FUNCTION_BLOCK TestRecieve EXTENDS Object IMPLEMENTS IDataReciever
VAR
    buffer : testData;
    currentLength : UDINT;
END_VAR

{attribute '''NORMAL__COMMENT' := ' New data recieved'}
(* New data recieved*)
METHOD NewDataRecieved : HResult
VAR_INPUT
	data	: Data; //Data recieved
END_VAR
IF currentLength + data.length > 9999 THEN
    currentLength := 0;
END_IF

Tc2_System.MEMCPY(destAddr := ADR(buffer.buffer[currentLength]),srcAddr := data.data, n := data.length); 

currentLength := currentLength + data.length;
END_METHOD

(*Reset error, allways call super*)
METHOD Reset
Tc2_System.MEMSET(destAddr := ADR(buffer), fillByte := 0, n := SIZEOF(buffer));
currentLength := 0;
END_METHOD

END_FUNCTION_BLOCK

(* stored: Version 1.1.0.1, ProductVersion 3.1.4020.12
   POU TestRecieve: Id {ac45b7df-f119-44bf-ad93-44d7bc6f8a02}, SpecialFunc None
   Method NewDataRecieved: Id {5380409a-4052-40e4-9eb6-8bd6a2573e60}
   Method Reset: Id {546fd031-9c6c-4eaf-92f6-be4c2cec096e} *)
